# EPICS substitutions: ek9000App/Db/EL2002_mbboDirect.substitutions
file EL2002.template
{       pattern
        {
                TERMINAL,

        }
        {
        }
}
